// TIA Portal V18 export
DATA_BLOCK "CMMS_Z2_FML_REF"   // DB69
{ S7_Optimized_Access := 'TRUE' }
VERSION : 0.1
// stored: AutoNumber true, DBAccessibleFromOPCUA true, IsOnlyStoredInLoadMemory false, IsRetainMemResEnabled false, IsWriteProtectedInAS false, MemoryReserve 100
   VAR
      FML_REF { S7_SetPoint := 'True'} : "DT_FML_REF";
   END_VAR
BEGIN
   FML_REF.DeviceType := 'CMMS';
END_DATA_BLOCK
